FUNCTION_BLOCK FB_Palletizer IMPLEMENTS ITF_Palletizer
VAR_INPUT
    // Alles komt later als echte units/interfaces. Nu alleen placeholders in comments.
    // RollerMotor       : ITF_Motor;            // elektro asynchroon motor (rollerband)
    // LiftServo         : ITF_Servo;            // servo ketting lift
    // Pin1              : ITF_LinearActuator;   // 4x pinnen
    // Pin2              : ITF_LinearActuator;
    // Pin3              : ITF_LinearActuator;
    // Pin4              : ITF_LinearActuator;
    // LsInfeed          : ITF_Lichtsensor;      // lichtsensor ingang
    // LsPosition        : ITF_Lichtsensor;      // lichtsensor einde/positie
    // DistanceFull      : ITF_Afstandssensor;   // opslag vol
    // DoorSensor        : ITF_DeurSensor;       // deur open sensor
    // LimitSwitch       : ITF_LimitSwitch;      // limit switch (positie onbekend)
    // EStop             : ITF_Noodstop;         // noodstop
    // OpenButton        : ITF_DrukKnop;         // open knop met licht
    // ResetButton       : ITF_DrukKnop;         // reset knop met licht
    // StatusLamp        : ITF_StatusLamp;       // machinestatuslamp
END_VAR

VAR
    // =========================
    // PackML command & status
    // =========================
    _CmdStatePal    : E_PackMLStates := E_PackMLStates.Idle;   // van control (1x trigger)
    _ActiveStatePal : E_PackMLStates := E_PackMLStates.Idle;   // interne actieve state
    CurrentStatePal : E_PackMLStates := E_PackMLStates.Idle;   // feedback naar control

    TriggerState : E_PackMLStates := E_PackMLStates.Idle;      // toegevoegd (zoals Depalletizer)
    VorigeInputState : E_PackMLStates := E_PackMLStates.Idle;  // toegevoegd

    // =========================
    // Alarm / safety (later)
    // =========================
    _AlarmActive : BOOL := FALSE;
    _AlarmCode   : UDINT := 0;
    _EStopOk     : BOOL := TRUE;    // later: EStop.Ok
    _DoorIsOpen   : BOOL := FALSE;   // later: DoorSensor.Open

    // =========================
    // Deur bediening (later)
    // =========================
    _DoorOpenRequest  : BOOL := FALSE;  // request vanuit control/HMI
    _DoorOpenAllowed  : BOOL := FALSE;  // berekend (later)

    // =========================
    // Proces signalen (later)
    // =========================
    _PalletAtInFeed    : BOOL := FALSE; // later: LsInfeed.Detect
    _PalletInPosition  : BOOL := FALSE; // later: LsPosition.Detect
    _StorageFull       : BOOL := FALSE; // later: DistanceFull.Full

    // Execute sequence (later)
    Step : INT := 0;

	//vanaf hier tijdelijke var door missende units
	RolbandAanUit : BOOL;
	LiftOmhoogYesNo : BOOL;
	LiftOmlaagYesNo : BOOL;

	Pin1UitYesNo : BOOL;
	Pin2UitYesNo : BOOL;
	Pin3UitYesNo : BOOL;
	Pin4UitYesNo : BOOL;

	// “feedback” die jij handmatig zet om steps door te laten lopen
	Pin1UitAangekomen : BOOL;
	Pin2UitAangekomen : BOOL;
	Pin3UitAangekomen : BOOL;
	Pin4UitAangekomen : BOOL;

	Pin1InAangekomen : BOOL;
	Pin2InAangekomen : BOOL;
	Pin3InAangekomen : BOOL;
	Pin4InAangekomen : BOOL;

	LiftBovenAangekomen : BOOL;
	LiftBenedenAangekomen : BOOL;
	//eind var
END_VAR

// 1) Latch command -> active (zodat 1x trigger genoeg is)
IF _CmdStatePal <> VorigeInputState THEN
    TriggerState := _CmdStatePal;
END_IF

VorigeInputState := _CmdStatePal;

// 2) Feedback state (wat ik NU aan het doen ben)
CurrentStatePal := TriggerState;

// 3) (optioneel) bereken deur-toestemming (nu nog simpel; later met echte voorwaarden)
_DoorOpenAllowed := _EStopOk AND (CurrentStatePal = E_PackMLStates.Idle OR CurrentStatePal = E_PackMLStates.Stopped OR CurrentStatePal = E_PackMLStates.Held OR CurrentStatePal = E_PackMLStates.Suspended);
// later (voorbeeld):
// _DoorOpenAllowed := _EStopOk AND (CurrentStatePal = E_PackMLStates.Idle OR CurrentStatePal = E_PackMLStates.Stopped OR CurrentStatePal = E_PackMLStates.Held OR CurrentStatePal = E_PackMLStates.Suspended);

// 4) PackML state machine (methods maak jij hierna aan)
CASE TriggerState OF

    E_PackMLStates.Idle:
        Idle();

    E_PackMLStates.Starting:
        Starting();

    E_PackMLStates.Execute:
        Execute();

    E_PackMLStates.Holding:
        Holding();

    E_PackMLStates.Held:
        Held();

    E_PackMLStates.Unholding:
        Unholding();

    E_PackMLStates.Suspending:
        Suspending();

    E_PackMLStates.Suspended:
        Suspended();

    E_PackMLStates.Unsuspending:
        Unsuspending();

    E_PackMLStates.Stopping:
        Stopping();

    E_PackMLStates.Stopped:
        Stopped();

    E_PackMLStates.Resetting:
        Resetting();

END_CASE

PROPERTY AlarmActive : BOOL
GET
AlarmActive := _AlarmActive;
END_GET
SET
_AlarmActive := AlarmActive;
END_SET
END_PROPERTY

PROPERTY AlarmCode : UDINT
GET
AlarmCode := _AlarmCode;
END_GET
SET
_AlarmCode := AlarmCode;
END_SET
END_PROPERTY

PROPERTY CurrentState : E_PackMLStates
GET
CurrentState := CurrentStatePal;
END_GET
SET
CurrentStatePal := CurrentState;
END_SET
END_PROPERTY

PROPERTY DoorIsOpen : BOOL
GET
DoorIsOpen := _DoorIsOpen;
END_GET
SET
_DoorIsOpen := DoorIsOpen;
END_SET
END_PROPERTY

PROPERTY DoorOpenAllowed : BOOL
GET
DoorOpenAllowed := _DoorOpenAllowed;
END_GET
SET
_DoorOpenAllowed := DoorOpenAllowed;
END_SET
END_PROPERTY

PROPERTY DoorOpenRequest : BOOL
GET
DoorOpenRequest := _DoorOpenRequest;
END_GET
SET
_DoorOpenRequest := DoorOpenRequest;
END_SET
END_PROPERTY

PROPERTY EStopOk : BOOL
GET
EStopOk := _EStopOk;
END_GET
SET
_EStopOk := EStopOk;
END_SET
END_PROPERTY

METHOD PUBLIC Execute : BOOL
CurrentStatePal := E_PackMLStates.Execute;

CASE Step OF

0:
	IF _PalletAtInFeed AND NOT _StorageFull THEN
		RolbandAanUit := TRUE;

		IF _PalletInPosition THEN
			RolbandAanUit := FALSE;
			Step := 10;
		END_IF
	ELSE
		RolbandAanUit := FALSE;
	END_IF


10:
	Pin1UitYesNo := TRUE;
	Pin2UitYesNo := TRUE;
	Pin3UitYesNo := TRUE;
	Pin4UitYesNo := TRUE;

	IF Pin1UitAangekomen AND Pin2UitAangekomen AND Pin3UitAangekomen AND Pin4UitAangekomen THEN
		Step := 20;
	END_IF


20:
	LiftOmhoogYesNo := TRUE;
	LiftOmlaagYesNo := FALSE;

	IF LiftBovenAangekomen THEN
		LiftOmhoogYesNo := FALSE;
		Step := 30;
	END_IF


30:
	Pin1UitYesNo := FALSE;
	Pin2UitYesNo := FALSE;
	Pin3UitYesNo := FALSE;
	Pin4UitYesNo := FALSE;

	IF Pin1InAangekomen AND Pin2InAangekomen AND Pin3InAangekomen AND Pin4InAangekomen THEN
		Step := 40;
	END_IF


40:
	LiftOmlaagYesNo := TRUE;
	LiftOmhoogYesNo := FALSE;

	IF LiftBenedenAangekomen THEN
		LiftOmlaagYesNo := FALSE;

		_PalletAtInFeed := FALSE;
		_PalletInPosition := FALSE;

		Step := 0;
	END_IF


ELSE
	Step := 0;
END_CASE

Execute := TRUE;
END_METHOD

METHOD PUBLIC Held : BOOL
CurrentStatePal := E_PackMLStates.Held;

RolbandAanUit := FALSE;
LiftOmhoogYesNo := FALSE;
LiftOmlaagYesNo := FALSE;

Held := TRUE;
END_METHOD

METHOD PUBLIC Holding : BOOL
CurrentStatePal := E_PackMLStates.Holding;

RolbandAanUit := FALSE;

LiftOmhoogYesNo := FALSE;
LiftOmlaagYesNo := FALSE;

TriggerState := E_PackMLStates.Held;

Holding := TRUE;
END_METHOD

METHOD PUBLIC Idle : BOOL
CurrentStatePal := E_PackMLStates.Idle;

RolbandAanUit := FALSE;

LiftOmhoogYesNo := FALSE;
LiftOmlaagYesNo := TRUE;

Pin1UitYesNo := FALSE;
Pin2UitYesNo := FALSE;
Pin3UitYesNo := FALSE;
Pin4UitYesNo := FALSE;

Step := 0;

Idle := TRUE;
END_METHOD

PROPERTY InputState : E_PackMLStates
GET
InputState := _CmdStatePal;
END_GET
SET
_CmdStatePal := InputState;
END_SET
END_PROPERTY

PROPERTY PalletAtInFeed : BOOL
GET
PalletAtInFeed := _PalletAtInFeed;
END_GET
SET
_PalletAtInFeed := PalletAtInFeed;
END_SET
END_PROPERTY

PROPERTY PalletInPosition : BOOL
GET
PalletInPosition := _PalletInPosition;
END_GET
SET
_PalletInPosition := PalletInPosition;
END_SET
END_PROPERTY

METHOD PUBLIC Resetting : BOOL
CurrentStatePal := E_PackMLStates.Resetting;

Step := 0;
_AlarmActive := FALSE;
_AlarmCode := 0;

TriggerState := E_PackMLStates.Idle;

Resetting := TRUE;
END_METHOD

METHOD PUBLIC Starting : BOOL
CurrentStatePal := E_PackMLStates.Starting;

RolbandAanUit := FALSE;

LiftOmlaagYesNo := TRUE;
LiftOmhoogYesNo := FALSE;

Pin1UitYesNo := FALSE;
Pin2UitYesNo := FALSE;
Pin3UitYesNo := FALSE;
Pin4UitYesNo := FALSE;

IF  _EStopOk AND NOT _DoorIsOpen AND
	LiftBenedenAangekomen AND
	Pin1InAangekomen AND Pin2InAangekomen AND Pin3InAangekomen AND Pin4InAangekomen
THEN
	TriggerState := E_PackMLStates.Execute;
	Step := 0;
END_IF

Starting := TRUE;
END_METHOD

METHOD PUBLIC Stopped : BOOL
CurrentStatePal := E_PackMLStates.Stopped;

RolbandAanUit := FALSE;
LiftOmhoogYesNo := FALSE;
LiftOmlaagYesNo := FALSE;

Stopped := TRUE;
END_METHOD

METHOD PUBLIC Stopping : BOOL
CurrentStatePal := E_PackMLStates.Stopping;

RolbandAanUit := FALSE;
LiftOmhoogYesNo := FALSE;
LiftOmlaagYesNo := FALSE;

TriggerState := E_PackMLStates.Stopped;

Stopping := TRUE;
END_METHOD

PROPERTY StorageFull : BOOL
GET
StorageFull := _StorageFull;
END_GET
SET
_StorageFull := StorageFull;
END_SET
END_PROPERTY

METHOD PUBLIC Suspended : BOOL
CurrentStatePal := E_PackMLStates.Suspended;

RolbandAanUit := FALSE;
LiftOmhoogYesNo := FALSE;
LiftOmlaagYesNo := FALSE;

Suspended := TRUE;
END_METHOD

METHOD PUBLIC Suspending : BOOL
CurrentStatePal := E_PackMLStates.Suspending;

RolbandAanUit := FALSE;
LiftOmhoogYesNo := FALSE;
LiftOmlaagYesNo := FALSE;

TriggerState := E_PackMLStates.Suspended;

Suspending := TRUE;
END_METHOD

METHOD PUBLIC Unholding : BOOL
CurrentStatePal := E_PackMLStates.Unholding;

TriggerState := E_PackMLStates.Execute;

Unholding := TRUE;
END_METHOD

METHOD PUBLIC Unsuspending : BOOL
CurrentStatePal := E_PackMLStates.Unsuspending;

TriggerState := E_PackMLStates.Execute;

Unsuspending := TRUE;
END_METHOD

END_FUNCTION_BLOCK

(* stored: Version 1.1.0.1
   POU FB_Palletizer: Id {01892087-3837-44fd-a643-766816d2ad24}, SpecialFunc None
   Folder Methods: Id {2411fb30-dde0-4d1e-a72d-103cc5262fde}
   Folder Properties: Id {f17e31d7-e075-4eb3-8dc3-3f972bfb1b56}
   Property AlarmActive: Id {d7b450da-7824-4bd0-81e2-c0a95cad9401}
   Get Get: Id {eca61404-5a79-4429-95f6-08988908187b}
   Set Set: Id {906ec274-904a-42e8-a9a8-b3a672975994}
   Property AlarmCode: Id {7775918f-adb8-440a-a083-a693ec6e35ed}
   Get Get: Id {bee063f1-d350-4cc0-9ddf-11a4c5476562}
   Set Set: Id {ca9637bc-d66f-4208-9988-26723f9017e8}
   Property CurrentState: Id {86f7f3c9-e77a-4903-966c-69e094622844}
   Get Get: Id {d21af37f-af47-40c7-9306-c35e3188c8cc}
   Set Set: Id {22c2287f-24b9-4ef4-bf61-4cc56975a5c7}
   Property DoorIsOpen: Id {63494c90-322d-4e57-8251-fba1448e45e3}
   Get Get: Id {1dfbb15f-9d04-4806-8b55-8787f8e62506}
   Set Set: Id {49730893-7421-4c3c-af1b-f4379f1f7258}
   Property DoorOpenAllowed: Id {c1dd9ef3-8cb6-40f3-b162-dd650ec12e30}
   Get Get: Id {f76b4f28-b3fc-4f08-b645-0fd36abcd3f3}
   Set Set: Id {d212a0f7-a7b6-4545-a555-9f085216c532}
   Property DoorOpenRequest: Id {0b451954-fb07-41ea-8774-059201d15865}
   Get Get: Id {6988e8a2-99a8-4038-b649-1043cde7c52a}
   Set Set: Id {374400ba-bd0b-4493-b00f-9bd286d247c2}
   Property EStopOk: Id {f31c760d-6c16-463a-9eca-26809f55fd3c}
   Get Get: Id {004a68f6-c794-41bf-8766-161c9ab2aa7d}
   Set Set: Id {8d171750-53fb-49e1-9f26-19141af429de}
   Method Execute: Id {16a58c6d-d9e6-4e7f-a0b7-9d7181b8bae5}
   Method Held: Id {b55bfaea-9ac2-400e-965a-9535331cf67e}
   Method Holding: Id {52861f9b-a481-4e23-b1c5-cef64c3ef4eb}
   Method Idle: Id {14dcf620-4eca-4676-82d0-855220591e82}
   Property InputState: Id {e710e0b2-3ee0-42cd-b804-7c79824640cd}
   Get Get: Id {56a237f1-68f6-40b0-bff6-449d06cb3f65}
   Set Set: Id {4be1caf8-933c-4f9d-8a71-87f693701266}
   Property PalletAtInFeed: Id {ba000df6-d778-49ce-bd26-d658733b31e3}
   Get Get: Id {8f14f7c4-34d5-4fc7-b4e1-a198e824f166}
   Set Set: Id {f8ddcfbc-e844-48ff-b381-0e6efae71e5b}
   Property PalletInPosition: Id {b0fe5337-b48e-4cd7-97dd-f88d45ce7267}
   Get Get: Id {02c129c5-a62d-44a7-94a0-16e435716629}
   Set Set: Id {0617f62a-eabd-43ca-94a1-4de5e38af927}
   Method Resetting: Id {db63cd78-6dfc-4b29-9463-c18ba5eaec19}
   Method Starting: Id {4a3e5953-84c4-41e7-a958-1b74ee60f666}
   Method Stopped: Id {33b48153-f3a7-47de-8cf8-6ac124fe3b32}
   Method Stopping: Id {cbd45afb-ba08-45da-9160-712941d6e40f}
   Property StorageFull: Id {d80f0c9b-02a2-425d-ad7e-65678d1810dd}
   Get Get: Id {1804146a-488c-464c-8d7b-8003a984bb2c}
   Set Set: Id {ad87cd23-966a-43c6-b2c0-c10a90a9a3f7}
   Method Suspended: Id {6a115e32-659e-43cc-88d2-1267419091bd}
   Method Suspending: Id {0dd5f12e-8033-42e3-9131-1e90a5f8e595}
   Method Unholding: Id {2351bdac-eb65-45f6-a51b-6a7044f90e63}
   Method Unsuspending: Id {1ee279d3-4eb2-48a5-ba89-aef09f4f2dbe} *)
